% RSLogix 500 project PRENSA_22MAYO2024.RSS, saved by version 8.40.00.08 %
PROJECT "UNTITLED"    % processor: MicroLogix 1400 %

PROGRAM FILES
  LAD 2 "SECUENCIA"  8 rungs
  LAD 3 "MANUAL"  3 rungs
  LAD 4 "OUTPUTS"  4 rungs
  LAD 5 "SEGURIDAD"  5 rungs

DATA FILES
  O0 OUTPUT  6 elements
  I1 INPUT  8 elements
  S2 STATUS  66 elements
  B3 BINARY  5 elements
  T4 TIMER  5 elements
  C5 COUNTER  1 elements
  R6 CONTROL  1 elements
  N7 INTEGER  1 elements
  F8 FLOAT  1 elements

LADDER 2 "SECUENCIA"
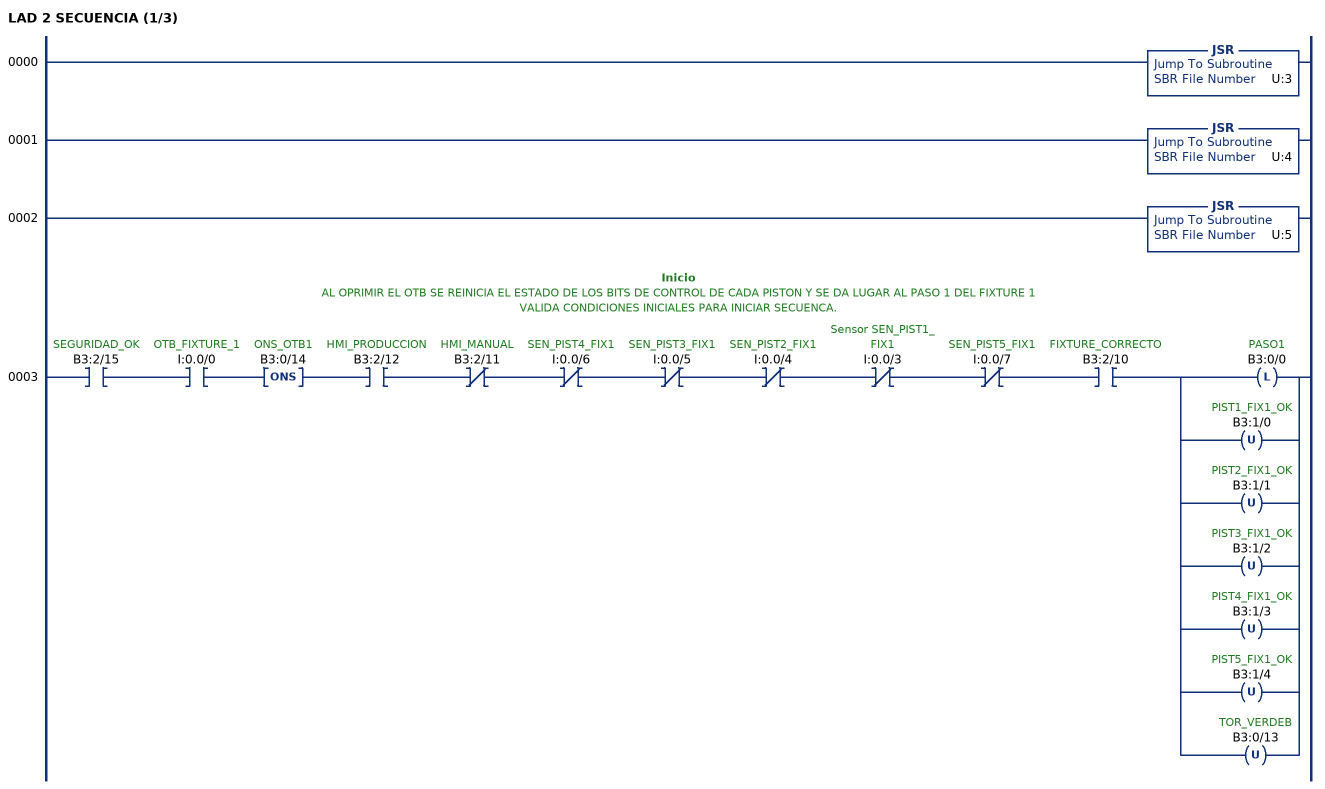
% Rung: 0 %
SOR JSR U:3 EOR
% Rung: 1 %
SOR JSR U:4 EOR
% Rung: 2 %
SOR JSR U:5 EOR
% Rung: 3 %
% TITLE: Inicio %
% AL OPRIMIR EL OTB SE REINICIA EL ESTADO DE LOS BITS DE CONTROL DE CADA PISTON Y SE DA LUGAR AL PASO 1 DEL FIXTURE 1
% VALIDA CONDICIONES INICIALES PARA INICIAR SECUENCA. %
SOR XIC B3:2/15 XIC I:0.0/0 ONS B3:0/14 XIC B3:2/12 XIO B3:2/11 XIO I:0.0/6 XIO I:0.0/5 XIO I:0.0/4 XIO I:0.0/3 XIO I:0.0/7 XIC B3:2/10 BST OTL B3:0/0 NXB OTU B3:1/0 NXB OTU B3:1/1 NXB OTU B3:1/2 NXB OTU B3:1/3 NXB OTU B3:1/4 NXB OTU B3:0/13 BND EOR
%   B3:2/15  SEGURIDAD_OK %
%   I:0.0/0  OTB_FIXTURE_1 %
%   B3:0/14  ONS_OTB1 %
%   B3:2/12  HMI_PRODUCCION %
%   B3:2/11  HMI_MANUAL %
%   I:0.0/6  SEN_PIST4_FIX1 %
%   I:0.0/5  SEN_PIST3_FIX1 %
%   I:0.0/4  SEN_PIST2_FIX1 %
%   I:0.0/3  SEN_PIST1_FIX1  "Sensor" %
%   I:0.0/7  SEN_PIST5_FIX1 %
%   B3:2/10  FIXTURE_CORRECTO %
%   B3:0/0  PASO1 %
%   B3:1/0  PIST1_FIX1_OK %
%   B3:1/1  PIST2_FIX1_OK %
%   B3:1/2  PIST3_FIX1_OK %
%   B3:1/3  PIST4_FIX1_OK %
%   B3:1/4  PIST5_FIX1_OK %
%   B3:0/13  TOR_VERDEB %

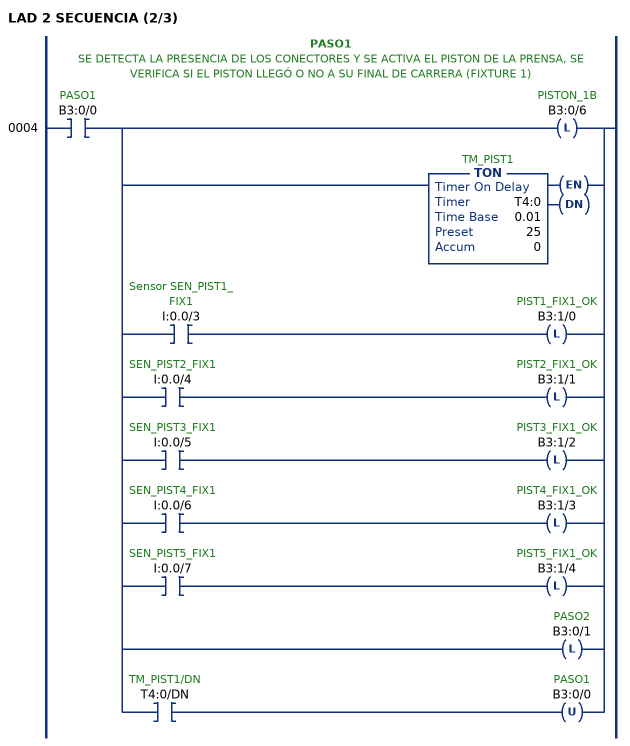
% Rung: 4 %
% TITLE: PASO1 %
% SE DETECTA LA PRESENCIA DE LOS CONECTORES Y SE ACTIVA EL PISTON DE LA PRENSA, SE VERIFICA SI EL PISTON LLEGÓ O NO A SU FINAL DE CARRERA (FIXTURE 1) %
SOR XIC B3:0/0 BST OTL B3:0/6 NXB TON T4:0 0.01 25 0 NXB XIC I:0.0/3 OTL B3:1/0 NXB XIC I:0.0/4 OTL B3:1/1 NXB XIC I:0.0/5 OTL B3:1/2 NXB XIC I:0.0/6 OTL B3:1/3 NXB XIC I:0.0/7 OTL B3:1/4 NXB OTL B3:0/1 NXB XIC T4:0/DN OTU B3:0/0 BND EOR
%   B3:0/0  PASO1 %
%   B3:0/6  PISTON_1B %
%   T4:0  TM_PIST1 %
%   I:0.0/3  SEN_PIST1_FIX1  "Sensor" %
%   B3:1/0  PIST1_FIX1_OK %
%   I:0.0/4  SEN_PIST2_FIX1 %
%   B3:1/1  PIST2_FIX1_OK %
%   I:0.0/5  SEN_PIST3_FIX1 %
%   B3:1/2  PIST3_FIX1_OK %
%   I:0.0/6  SEN_PIST4_FIX1 %
%   B3:1/3  PIST4_FIX1_OK %
%   I:0.0/7  SEN_PIST5_FIX1 %
%   B3:1/4  PIST5_FIX1_OK %
%   B3:0/1  PASO2 %

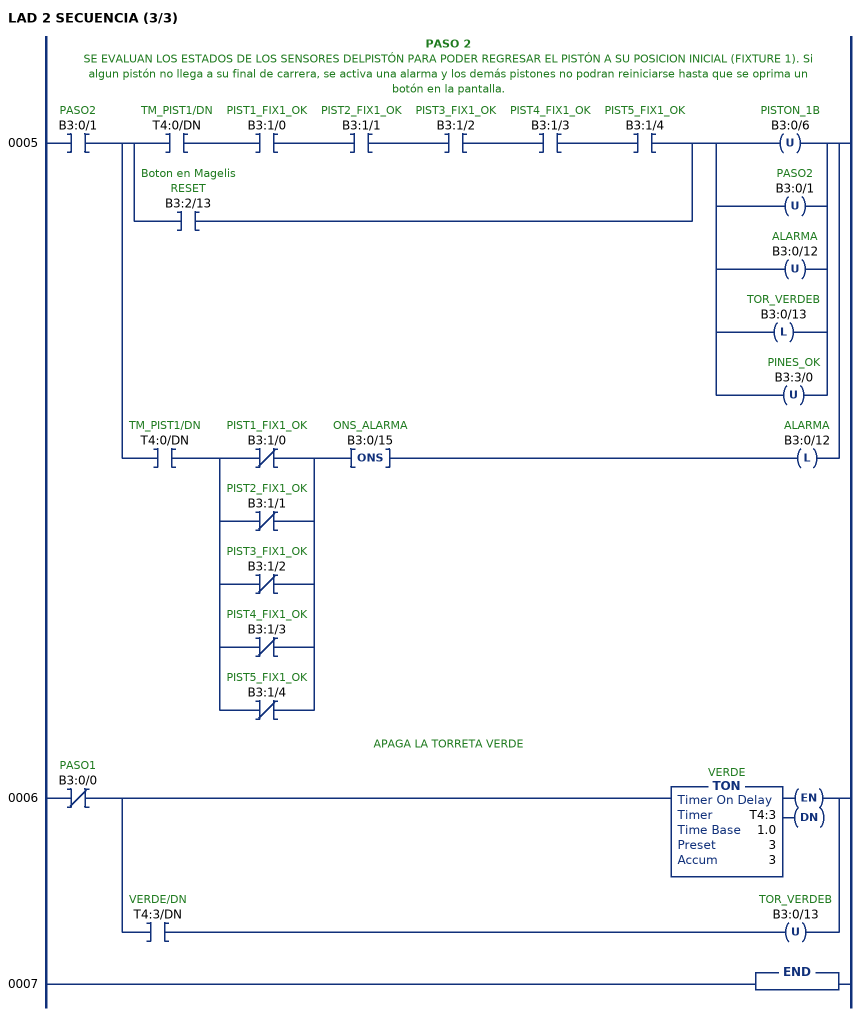
% Rung: 5 %
% TITLE: PASO 2 %
% SE EVALUAN LOS ESTADOS DE LOS SENSORES DELPISTÓN PARA PODER REGRESAR EL PISTÓN A SU POSICION INICIAL (FIXTURE 1). Si algun pistón no llega a su final de carrera, se activa una alarma y los demás pistones no podran reiniciarse hasta que se oprima un botón en la pantalla. %
SOR XIC B3:0/1 BST BST XIC T4:0/DN XIC B3:1/0 XIC B3:1/1 XIC B3:1/2 XIC B3:1/3 XIC B3:1/4 NXB XIC B3:2/13 BND BST OTU B3:0/6 NXB OTU B3:0/1 NXB OTU B3:0/12 NXB OTL B3:0/13 NXB OTU B3:3/0 BND NXB XIC T4:0/DN BST XIO B3:1/0 NXB XIO B3:1/1 NXB XIO B3:1/2 NXB XIO B3:1/3 NXB XIO B3:1/4 BND ONS B3:0/15 OTL B3:0/12 BND EOR
%   B3:0/1  PASO2 %
%   T4:0  TM_PIST1 %
%   B3:1/0  PIST1_FIX1_OK %
%   B3:1/1  PIST2_FIX1_OK %
%   B3:1/2  PIST3_FIX1_OK %
%   B3:1/3  PIST4_FIX1_OK %
%   B3:1/4  PIST5_FIX1_OK %
%   B3:2/13  RESET  "Boton en Magelis" %
%   B3:0/6  PISTON_1B %
%   B3:0/12  ALARMA %
%   B3:0/13  TOR_VERDEB %
%   B3:3/0  PINES_OK %
%   B3:0/15  ONS_ALARMA %
% Rung: 6 %
% APAGA LA TORRETA VERDE %
SOR XIO B3:0/0 BST TON T4:3 1.0 3 3 NXB XIC T4:3/DN OTU B3:0/13 BND EOR
%   B3:0/0  PASO1 %
%   T4:3  VERDE %
%   B3:0/13  TOR_VERDEB %
% Rung: 7 %
SOR END EOR

LADDER 3 "MANUAL"
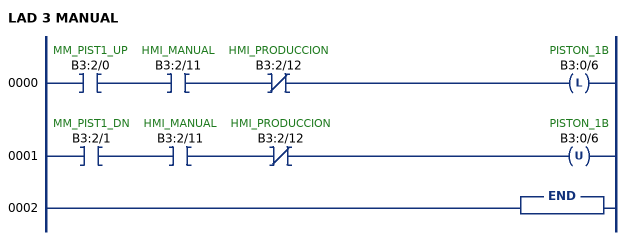
% Rung: 0 %
SOR XIC B3:2/0 XIC B3:2/11 XIO B3:2/12 OTL B3:0/6 EOR
%   B3:2/0  MM_PIST1_UP %
%   B3:2/11  HMI_MANUAL %
%   B3:2/12  HMI_PRODUCCION %
%   B3:0/6  PISTON_1B %
% Rung: 1 %
SOR XIC B3:2/1 XIC B3:2/11 XIO B3:2/12 OTU B3:0/6 EOR
%   B3:2/1  MM_PIST1_DN %
%   B3:2/11  HMI_MANUAL %
%   B3:2/12  HMI_PRODUCCION %
%   B3:0/6  PISTON_1B %
% Rung: 2 %
SOR END EOR

LADDER 4 "OUTPUTS"
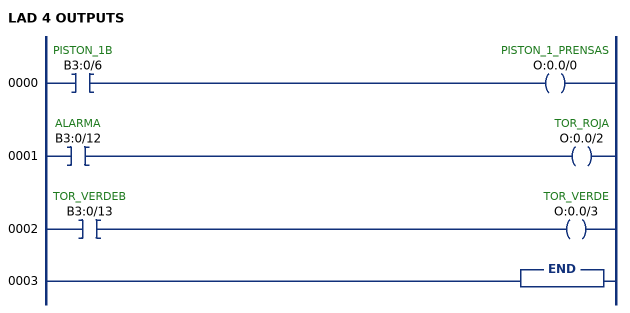
% Rung: 0 %
SOR XIC B3:0/6 OTE O:0.0/0 EOR
%   B3:0/6  PISTON_1B %
%   O:0.0/0  PISTON_1_PRENSAS %
% Rung: 1 %
SOR XIC B3:0/12 OTE O:0.0/2 EOR
%   B3:0/12  ALARMA %
%   O:0.0/2  TOR_ROJA %
% Rung: 2 %
SOR XIC B3:0/13 OTE O:0.0/3 EOR
%   B3:0/13  TOR_VERDEB %
%   O:0.0/3  TOR_VERDE %
% Rung: 3 %
SOR END EOR

LADDER 5 "SEGURIDAD"
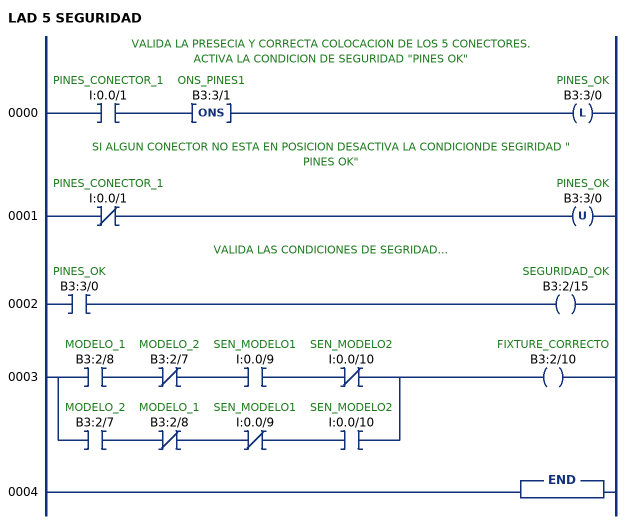
% Rung: 0 %
% VALIDA LA PRESECIA Y CORRECTA COLOCACION DE LOS 5 CONECTORES.
% ACTIVA LA CONDICION DE SEGURIDAD "PINES OK" %
SOR XIC I:0.0/1 ONS B3:3/1 OTL B3:3/0 EOR
%   I:0.0/1  PINES_CONECTOR_1 %
%   B3:3/1  ONS_PINES1 %
%   B3:3/0  PINES_OK %
% Rung: 1 %
% SI ALGUN CONECTOR NO ESTA EN POSICION DESACTIVA LA CONDICIONDE SEGIRIDAD " PINES OK" %
SOR XIO I:0.0/1 OTU B3:3/0 EOR
%   I:0.0/1  PINES_CONECTOR_1 %
%   B3:3/0  PINES_OK %
% Rung: 2 %
% VALIDA LAS CONDICIONES DE SEGRIDAD... %
SOR XIC B3:3/0 OTE B3:2/15 EOR
%   B3:3/0  PINES_OK %
%   B3:2/15  SEGURIDAD_OK %
% Rung: 3 %
SOR BST XIC B3:2/8 XIO B3:2/7 XIC I:0.0/9 XIO I:0.0/10 NXB XIC B3:2/7 XIO B3:2/8 XIO I:0.0/9 XIC I:0.0/10 BND OTE B3:2/10 EOR
%   B3:2/8  MODELO_1 %
%   B3:2/7  MODELO_2 %
%   I:0.0/9  SEN_MODELO1 %
%   I:0.0/10  SEN_MODELO2 %
%   B3:2/10  FIXTURE_CORRECTO %
% Rung: 4 %
SOR END EOR

OTHER DOCUMENTED ADDRESSES
  B3:0/2  PASO3
  B3:0/3  PASO1_2
  B3:0/4  PASO2_2
  B3:0/7  ACTIVAR_CANDADO
  B3:0/8  PISTON_3B
  B3:0/9  PASO1_3
  B3:0/10  PASO2_3
  B3:1/5  PIST1_FIX2_OK
  B3:1/6  PIST2_FIX2_OK
  B3:1/7  PIST3_FIX2_OK
  B3:1/8  PIST4_FIX2_OK
  B3:1/9  PIST5_FIX2_OK
  B3:1/10  PIST1_FIX3_OK
  B3:1/11  PIST2_FIX3_OK
  B3:1/12  PIST3_FIX3_OK
  B3:1/13  PIST4_FIX3_OK
  B3:1/14  PIST5_FIX3_OK
  B3:2/4  MM_PIST3_UP
  B3:2/5  VALIDAR_SENSOR2
  B3:2/6  VALIDAR_SENSOR1
  B3:2/9  GUIA_CABLES_OK
  B3:2/14  MAG_OK
  B3:3/2  ONS_PINES2
  B3:3/3  PINES2_OK
  B3:3/4  ONS_OTB2
  B3:3/5  TOR_VERDE2B
  B3:3/6  ALARMA2
  B3:3/7  ONS_ALARMA2
  B3:3/8  RESET2
  I:0.0/2  SEN_PRESION
  I:0.0/8  SENSOR_CANDADO_FIX1
  I:1.0/6  SEN_PIST1_FIX2
  I:1.0/7  SEN_PIST2_FIX2
  I:1.0/8  SEN_PIST3_FIX2
  I:1.0/9  SEN_PIST4_FIX2
  I:1.0/10  SEN_PIST5_FIX2
  I:1.0/11  SEN_PIST1_FIX3
  I:1.0/12  SEN_PIST2_FIX3
  I:1.0/13  SEN_PIST3_FIX3
  I:1.0/14  SEN_PIST4_FIX3
  I:1.0/15  SEN_PIST5_FIX3
  O:0.0/1  PISTON_2_CANDADO
  O:0.0/5  TOR2_VERDE
  T4:1  TM_PIST2
  T4:2  TM_PIST3
  T4:4  VERDE2

COMMENTS NOT ATTACHED TO A CURRENT RUNG
  B3:0/1: PASO 2
  B3:0/10: PASO 1 FIXTURE 3 / SE DETECTA LA PRESENCIA DE LOS CONECTORES Y SE ACTIVA EL PISTON DE LA PRENSA, SE VERIFICA SI EL PISTON LLEGÓ O NO A SU FINAL DE CARRERA
  B3:0/4: PASO 1 FIXTURE 2 / SE DETECTA LA PRESENCIA DE LOS CONECTORES Y SE ACTIVA EL PISTON DE LA PRENSA, SE VERIFICA SI EL PISTON LLEGÓ O NO A SU FINAL DE CARRERA
  B3:0/0: PASO1 FIXTURE 1 / SE DETECTA LA PRESENCIA DE LOS CONECTORES Y SE ACTIVA EL PISTON DE LA PRENSA, SE VERIFICA SI EL PISTON LLEGÓ O NO A SU FINAL DE CARRERA
  B3:1/4: AL OPRIMIR EL OTB SE REINICIA EL ESTADO DE LOS BITS DE CONTROL DE CADA PISTON Y SE DA LUGAR AL PASO 1 DEL FIXTURE 2

REVISION NOTES
  0: Actualizacion 21/02/2024

DATA TABLE (non-zero values as saved)
DATA B3
% B3:0 % 0X0010 0X003F 0XC000 0X0043 0X0000
DATA T4
% .PRE .ACC %
% T4:0 % 25 0
% T4:1 % 25 0
% T4:2 % 100 0
% T4:3 % 3 3
% T4:4 % 3 3
